(* Logix 5000 project; controller EuniceF_Lab2 vendor 1 type 14 code 150 rev 37.11; software revision 37.00 *)

TASK MainTask (continuous, watchdog 500 ms) : MainProgram

MODULES
   Local : vendor 1 type 14 code 150 (Compact 0, rev 37.11)
      Discrete_IO : Embedded (Compact 1, rev 3.1, Output RPI 20 ms)
      Analog_IO : Embedded (Compact 2, rev 1.1, Output RPI 80 ms)
      Counters : Embedded (Compact 3, rev 1.1, Output RPI 20 ms)
END_MODULES

VAR_GLOBAL   (* controller tags *)
   Diif_Pressure : ALIAS FOR Local:2:I.Ch3Data;
   DrainClose : DINT;
   DrainValve : ALIAS FOR Local:1:O.Data.10;
   Height : REAL;
   HSC_Enable : ALIAS FOR Local:3:O.Ctr0En;
   HSC_Reset : ALIAS FOR Local:3:O.Ctr0SoftPreset;
   Kfactor : DINT;
   Mixer : ALIAS FOR Local:1:O.Data.9;
   Pump : ALIAS FOR Local:1:O.Data.8;
   Start : ALIAS FOR Local:1:I.Data.11;
   Stop : ALIAS FOR Local:1:I.Data.9;
   T1 : TIMER := (PRE := 10000);
   Value : ALIAS FOR Local:2:I.Ch0Data;
   Valve_Position : ALIAS FOR Local:2:O.Ch1Data;
END_VAR

PROGRAM MainProgram   (* main routine MainRoutine *)
VAR
   Seq1 : DINT;
END_VAR

ROUTINE MainRoutine   (* ladder *)
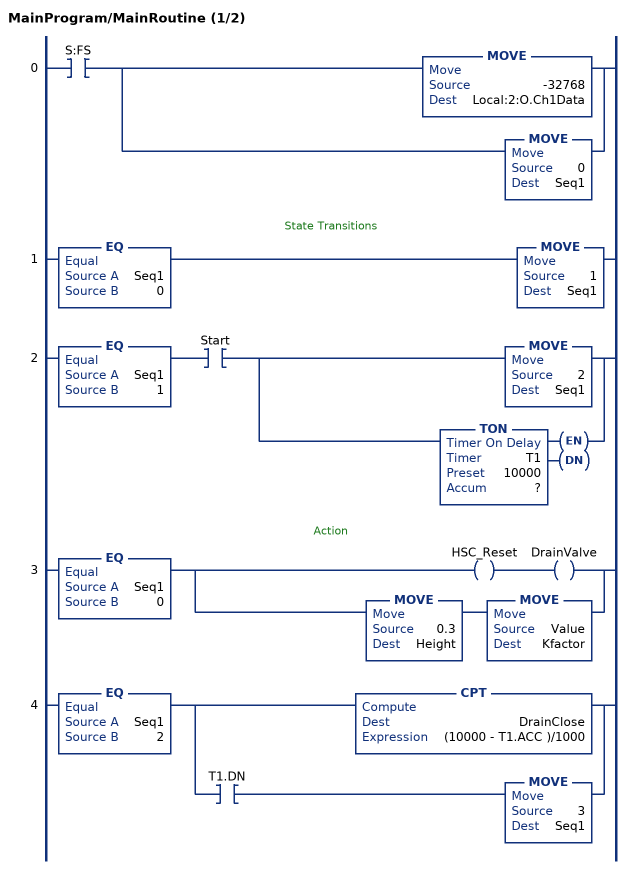
   0: XIC(S:FS)[MOVE(-32768,Local:2:O.Ch1Data) ,MOVE(0,Seq1) ];
   // State Transitions
   1: EQ(Seq1,0)MOVE(1,Seq1);
   2: EQ(Seq1,1)XIC(Start)[MOVE(2,Seq1) ,TON(T1,?,?) ];
   // Action
   3: EQ(Seq1,0)[OTE(HSC_Reset) OTE(DrainValve) ,MOVE(0.3,Height) MOVE(Value,Kfactor) ];
   4: EQ(Seq1,2)[CPT(DrainClose,(10000 - T1.ACC )/1000) ,XIC(T1.DN) MOVE(3,Seq1) ];
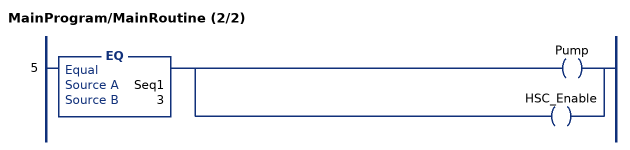
   5: EQ(Seq1,3)[OTE(Pump) ,OTE(HSC_Enable) ];
END_ROUTINE
END_PROGRAM
